{attribute 'qualified_only'}
VAR_GLOBAL
 	fSimulationTime : LREAL; 
	fCylinderVelocityReference : LREAL; 
	fBoomAngleDeg : LREAL;
	fMaxPistonPosition : LREAL;
	sPistonEndStopMessages : STRING;
	bOn : BOOL;
	bAuto : BOOL;
	bPowerOn : BOOL;
	bStart : BOOL;
	bStop : BOOL;
	bRunning : BOOL;
	eMode : E_Mode;
	fManualCylinderPositionReference : LREAL; 
	fCylinderPosition : LREAL; 
	fCylinderPositionRestricted : LREAL; 
	stPistonAnimation : ST_RelativeMovement;
	stBoomAnimation : ST_RelativeMovement;
	eStatus : E_Status;
END_VAR

(* stored: Version 1.1.0.1, ProductVersion 3.1.4024.10
   GVL HMI: Id {515f7d22-94cb-4f67-80c3-c968411175ad} *)
